# EPICS autosave request: softglue/softGlueApp/Db/softGlue_FPGAContent_s1ID_Vgate_settings.req
# up/dn counters
file UpDnCntr_settings.req P=$(P),H=$(H),N=1
file UpDnCntr_settings.req P=$(P),H=$(H),N=2
